// TIA Portal V16 export
// export: Created 2023-01-03T15:35:07.6134871Z, ExportSetting WithDefaults, DisplayName Totally Integrated Automation Portal, DisplayVersion V16, DisplayName TIA Portal Version Control Interface, DisplayVersion V16, DisplayName TIA Portal Openness, DisplayVersion V16, DisplayName STEP 7 Professional, DisplayVersion V16, DisplayName STEP 7 Safety, DisplayVersion V16, DisplayName WinCC Advanced, DisplayVersion V16
FUNCTION_BLOCK "CYLINDER_AUTO"   // FB1, LAD
{ S7_Optimized_Access := 'TRUE' }
VERSION : 0.1
// stored: AutoNumber true, IsIECCheckEnabled false, IsRetainMemResEnabled false, MemoryReserve 100, SetENOAutomatically false, UDAEnableTagReadback false
BEGIN

REGION Network 1: cylinder -M4 extend
   // IF PART IS DETECTED AND MOTOR IS STOPPED AND CYLINDER IS NOT EXTENDED ALREADY, EXTEND THE CYLINDER
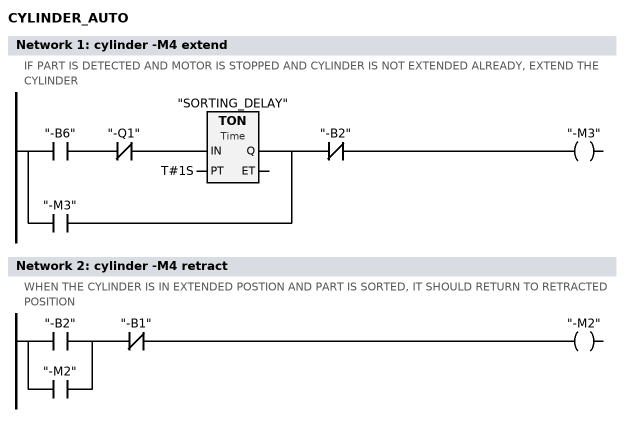
   RUNG wire#powerrail
      Contact( "-B6" )
      I_Contact( "-Q1" )
      { S7_Templates := "time_type := Time" } "SORTING_DELAY".TON(pt := T#1S, et =>)
      wire#w1
      I_Contact( "-B2" )
      Coil( "-M3" )
   END_RUNG
   RUNG wire#powerrail
      Contact( "-M3" )
   END_RUNG wire#w1
   // the same network as SCL:
   "SORTING_DELAY".TON(IN := "-B6" AND NOT "-Q1", PT := T#1S);
   "-M3" := ("SORTING_DELAY".Q OR "-M3") AND NOT "-B2";
END_REGION

REGION Network 2: cylinder -M4 retract
   // WHEN THE CYLINDER IS IN EXTENDED POSTION AND PART IS SORTED, IT SHOULD RETURN TO RETRACTED POSITION
   RUNG wire#powerrail
      Contact( "-B2" )
      wire#w1
      I_Contact( "-B1" )
      Coil( "-M2" )
   END_RUNG
   RUNG wire#powerrail
      Contact( "-M2" )
   END_RUNG wire#w1
   // the same network as SCL:
   "-M2" := ("-B2" OR "-M2") AND NOT "-B1";
END_REGION
END_FUNCTION_BLOCK
